TYPE TLoaderHead :
	(
		LH_Head1 := 0,
		LH_Head2
	);
END_TYPE

(* stored: Version 1.1.0.1, ProductVersion 3.1.4022.12
   DUT TLoaderHead: Id {c92a68f5-b6e7-4384-ae2a-8d5f2638d6b7} *)
